TYPE ST_STATION_LIST_RESULT :
STRUCT
  wState    : WORD;   // wState == 0 --> all ok
  nIndex    : ULINT;
  stData    : ST_STATION_MOVER_DATA;  // copy of list entry
END_STRUCT
END_TYPE

(* stored: Version 1.1.0.1, ProductVersion 3.1.4026.18
   DUT ST_STATION_LIST_RESULT: Id {bd4e306d-dfbd-47fc-b49f-859587a5b356} *)
